TYPE Cnv_Motor_DUT :
STRUCT
	Enable:	BOOL;
	Enabled:	BOOL;
	Ready:	BOOL;
	Forward:	BOOL;
	Reverse:	BOOL;
	Speed:	REAL;
	Speed_Actual:	REAL;
	Actual_Current:	REAL;
	Actual_Torque:	UINT;
	Config_Axis:	WORD;
	Error:	BOOL;
	Status:	WORD;
	Communication_Error:	WORD;
	Lockout:	BOOL;
END_STRUCT
END_TYPE

(* stored: Version 1.1.0.1
   DUT Cnv_Motor_DUT: Id {b142180c-abaf-4490-b433-f6d2125fe9be} *)
